// SIMATIC S7-200 SMART project (STEP 7-Micro/WIN SMART), CPU ST60

SYMBOL_TABLE V区符号
参数传输成功           V0.0     // 接收工控机传来的数据传输成功信号
参数是否更新           V0.1
挡板自动控制完成标志       V0.2
挡板电机开关           V0.3
挡板手动向内           V0.4
挡板手动向外           V0.5
置工件就绪            V1000.0
下料电机开关           V0.7
下料前进点动           V1.0
下料后退点动           V1.1
冷却电机开关           V1.2
冷却电机点动向内         V1.3
冷却电机点动向外         V1.4
挡板电机手动运行         V10.0
冷却电机手动运行         V10.1
下料电机手动运行         V10.2
挡板手动一键调节         V10.3
挡板一键调节完成标志       V10.4
挡板点动向内           V10.5
挡板点动向外           V10.6
挡板电机查找原点按钮       V11.1
下料电机查找原点按钮       V11.2
冷却电机查找原点按钮       V11.3
挡板自动控制           V11.4
下料下移一个工位         V11.5
下料启动按钮           V11.6
下料手动完成标志         V11.7
回到底部             V12.0
冷却自动控制           V12.1
挡板电机查找原点         V12.2
下料电机查找原点         V12.3
冷却电机查找原点         V12.4
冷却点动向内           V12.5
冷却点动向外           V12.6
挡板电机函数完成标志位      V20.1
挡板电机当前运动方向       V20.2
挡板电机查找原点完成位      V20.3
挡板电机GOTO完成位      V20.4
挡板电机错误参数         VB21
挡板电机当前位置         VD24
挡板电机当前速度         VD28
挡板电机移动位置         VD44
挡板电机速度           VD48
挡板电机移动模式         VB41
挡板电机停止运动轴        V40.1
挡板电机运动方向         V40.2
冷却电机初始化完成位       V60.1
冷却电机当前运动方向       V60.2
冷却电机查找原点完成位      V60.3
冷却电机GOTO完成位      V60.4
冷却电机错误参数         VB61
冷却电机当前位置         VD64
冷却电机当前速度         VD68
冷却电机移动位置         VD84
冷却电机速度           VD88
冷却电机移动模式         VB81
冷却电机停止运动轴        V80.1
冷却电机运动方向         V80.2
下料电机函数完成标志位      V100.1
下料电机当前运动方向       V100.2
下料电机查找原点完成位      V100.3
下料电机GOTO完成位      V100.4
下料电机错误参数         VB101
下料电机当前位置         VD104
下料电机当前速度         VD108
下料电机移动位置         VD124
下料电机速度           VD128
下料电机移动模式         VB121
下料电机停止运动轴        V120.1
下料电机运动方向         V120.2
下料电机运动到杆件放置      VD150
下料电机下移一个杆件位      VD154
下料电机一号杆件位置       VD158
下料电机二号杆件位置       VD162
下料电机三号杆件位置       VD166
下料电机四号杆件位置       VD170
下料电机五号杆件位置       VD174
下料电机运动到下料位置      VD178
上一杆件数据           VD140
当前杆件数据           VD144
轴0运动组态用          VB200    // VB200-VB292为轴0占用
轴1运动组态用          VB293    // VB293-VB385为轴1占用
轴2运动组态用          VB386    // VB386-VB478为轴2占用
链传动使能按钮          V400.0
链传动低速按钮          V400.1
链传动高速按钮          V400.2
链传动一个工位按钮        V400.3   // 链传动机构运动一个杆位按钮
链传动自动运行          V400.4
END_SYMBOL_TABLE

SYMBOL_TABLE 系统符号
Always_On        SM0.0    // 始终接通
First_Scan_On    SM0.1    // 仅在第一个扫描周期时接通
END_SYMBOL_TABLE

SYMBOL_TABLE M区符号
挡板超限报警           M0.0     // 挡板的位置超过左右极限传感器的位置
更新配对表            M0.1
电机是否就绪状态位        M0.3
上料步进到位状态位        M0.4
上料工件有无状态位        M0.5
下料步进到位状态位        M0.6
下料小车到位状态位        M0.7
步进报警信息           M1.0
上料传动故障报警         M1.1
两次杆件之差           MD12
END_SYMBOL_TABLE

SYMBOL_TABLE 定时器符号
顺序控制延时1          T33      // 短延时，保证正确读取到判断工件有无传感器的状态
顺序控制延时2          T34      // 短延时，保证正确读取到判断工件是否到位传感器的状态
顺序控制延时3          T35      // 短延时，保证正确读取到判断工件有无传感器的状态
上料故障报警定时         T37      // 设置定时，超时则报警
链传动控制定时器         T97
挡板运动脉冲1          T101     // 给一个运动脉冲信号，挡板移动到杆件长度处
下料运动脉冲1          T102     // 给一个运动脉冲信号，小车移动到机器人放料处
END_SYMBOL_TABLE

ORGANIZATION_BLOCK 主程序:OB1
TITLE=
BEGIN
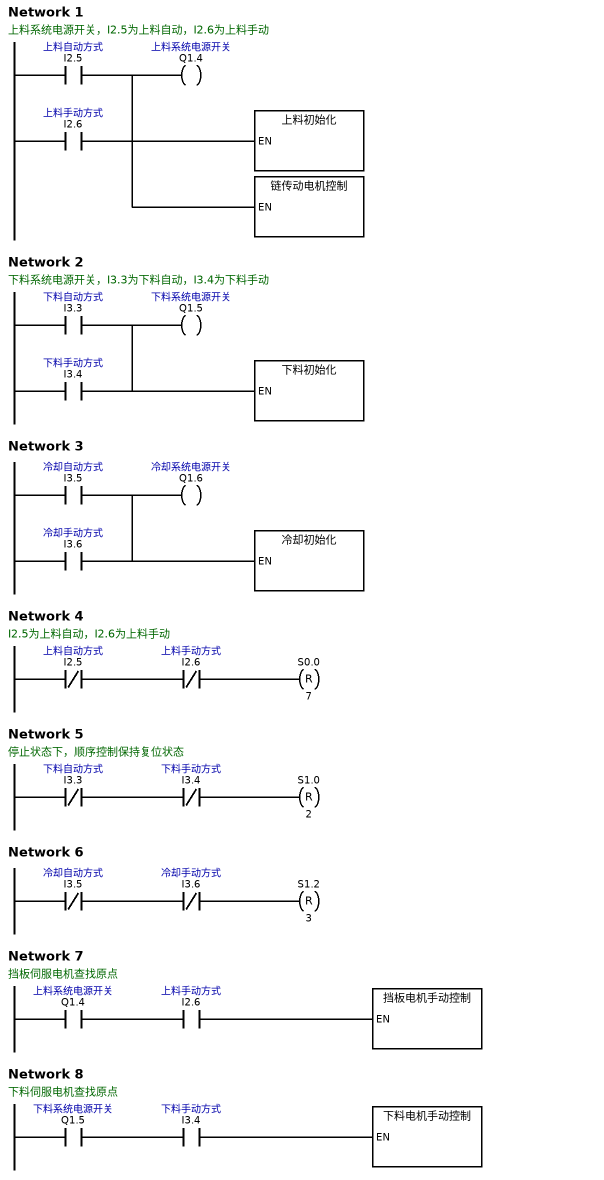
Network 1
// 上料系统电源开关，I2.5为上料自动，I2.6为上料手动
LD     上料自动方式:I2.5
O      上料手动方式:I2.6
=      上料系统电源开关:Q1.4
CALL   上料初始化:SBR14
CALL   链传动电机控制:SBR19
Network 2
// 下料系统电源开关，I3.3为下料自动，I3.4为下料手动
LD     下料自动方式:I3.3
O      下料手动方式:I3.4
=      下料系统电源开关:Q1.5
CALL   下料初始化:SBR15
Network 3
LD     冷却自动方式:I3.5
O      冷却手动方式:I3.6
=      冷却系统电源开关:Q1.6
CALL   冷却初始化:SBR16
Network 4
// I2.5为上料自动，I2.6为上料手动
LDN    上料自动方式:I2.5
AN     上料手动方式:I2.6
R      S0.0, 7
Network 5
// 停止状态下，顺序控制保持复位状态
LDN    下料自动方式:I3.3
AN     下料手动方式:I3.4
R      S1.0, 2
Network 6
LDN    冷却自动方式:I3.5
AN     冷却手动方式:I3.6
R      S1.2, 3
Network 7
// 挡板伺服电机查找原点
LD     上料系统电源开关:Q1.4
A      上料手动方式:I2.6
CALL   挡板电机手动控制:SBR7
Network 8
// 下料伺服电机查找原点
LD     下料系统电源开关:Q1.5
A      下料手动方式:I3.4
CALL   下料电机手动控制:SBR9
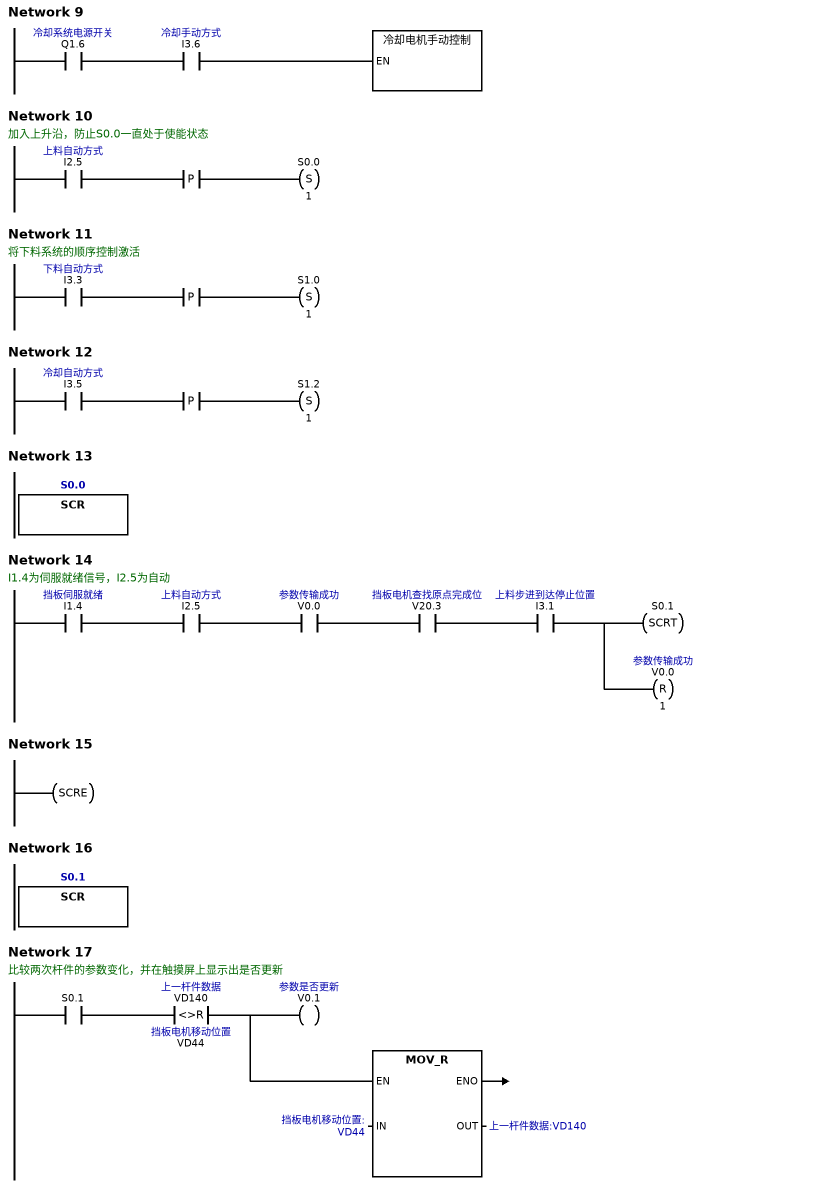
Network 9
LD     冷却系统电源开关:Q1.6
A      冷却手动方式:I3.6
CALL   冷却电机手动控制:SBR18
Network 10
// 加入上升沿，防止S0.0一直处于使能状态
LD     上料自动方式:I2.5
EU
S      S0.0, 1
Network 11
// 将下料系统的顺序控制激活
LD     下料自动方式:I3.3
EU
S      S1.0, 1
Network 12
LD     冷却自动方式:I3.5
EU
S      S1.2, 1
Network 13
LSCR   S0.0
Network 14
// I1.4为伺服就绪信号，I2.5为自动
LD     挡板伺服就绪:I1.4
A      上料自动方式:I2.5
A      参数传输成功:V0.0
A      挡板电机查找原点完成位:V20.3
A      上料步进到达停止位置:I3.1
SCRT   S0.1
R      参数传输成功:V0.0, 1
Network 15
SCRE
Network 16
LSCR   S0.1
Network 17
// 比较两次杆件的参数变化，并在触摸屏上显示出是否更新
LD     S0.1
AR<>   上一杆件数据:VD140, 挡板电机移动位置:VD44
=      参数是否更新:V0.1
MOVR   挡板电机移动位置:VD44, 上一杆件数据:VD140
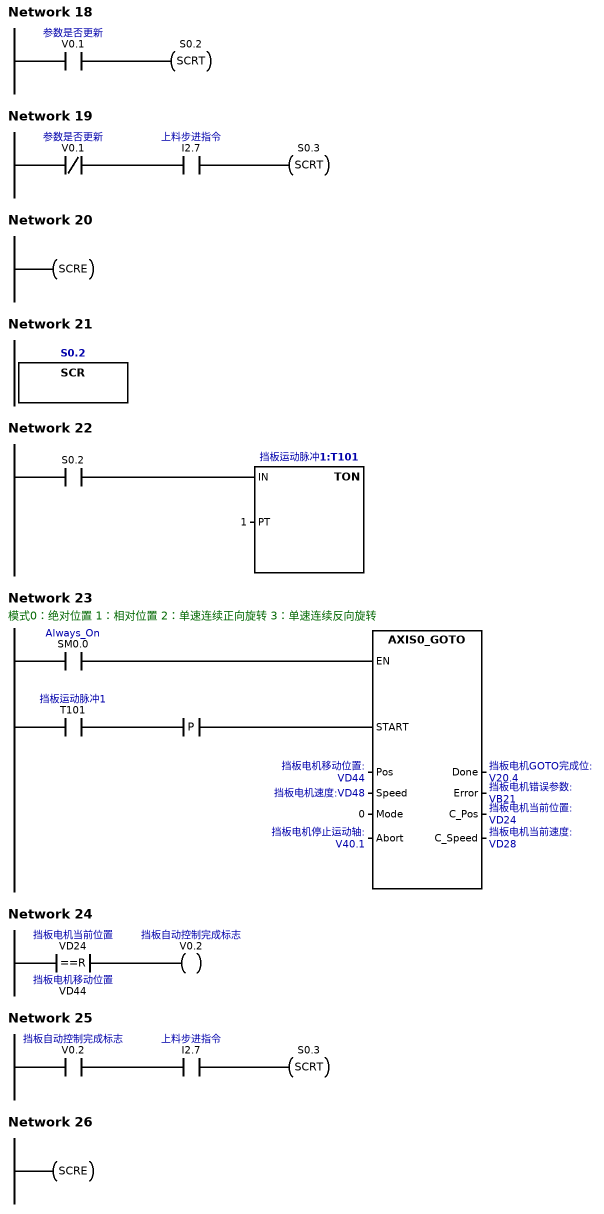
Network 18
LD     参数是否更新:V0.1
SCRT   S0.2
Network 19
LDN    参数是否更新:V0.1
A      上料步进指令:I2.7
SCRT   S0.3
Network 20
SCRE
Network 21
LSCR   S0.2
Network 22
LD     S0.2
TON    挡板运动脉冲1:T101, 1
Network 23
// 模式0：绝对位置 1：相对位置 2：单速连续正向旋转 3：单速连续反向旋转
LD     Always_On:SM0.0
=      L60.0
LD     挡板运动脉冲1:T101
EU
=      L63.7
LD     L60.0
CALL   AXIS0_GOTO:SBR2, L63.7, 挡板电机移动位置:VD44, 挡板电机速度:VD48, 0, 挡板电机停止运动轴:V40.1, 挡板电机GOTO完成位:V20.4, 挡板电机错误参数:VB21, 挡板电机当前位置:VD24, 挡板电机当前速度:VD28
Network 24
LDR=   挡板电机当前位置:VD24, 挡板电机移动位置:VD44
=      挡板自动控制完成标志:V0.2
Network 25
LD     挡板自动控制完成标志:V0.2
A      上料步进指令:I2.7
SCRT   S0.3
Network 26
SCRE
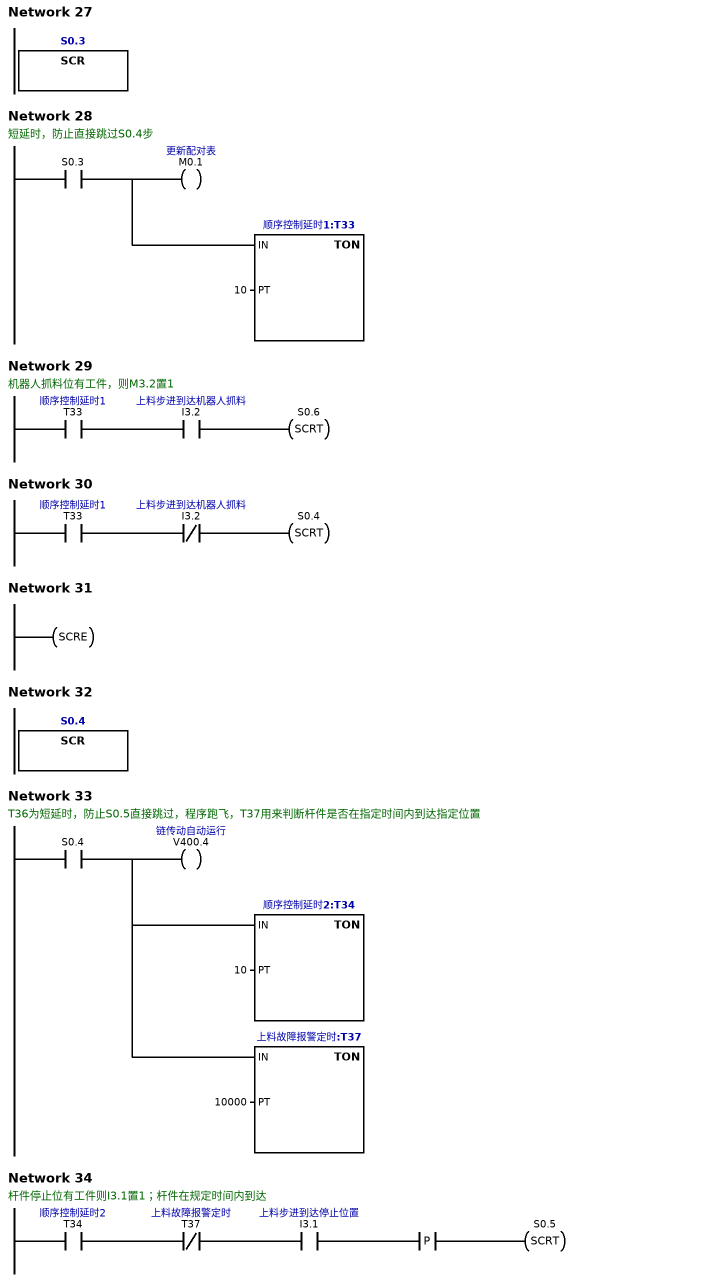
Network 27
LSCR   S0.3
Network 28
// 短延时，防止直接跳过S0.4步
LD     S0.3
=      更新配对表:M0.1
TON    顺序控制延时1:T33, 10
Network 29
// 机器人抓料位有工件，则M3.2置1
LD     顺序控制延时1:T33
A      上料步进到达机器人抓料:I3.2
SCRT   S0.6
Network 30
LD     顺序控制延时1:T33
AN     上料步进到达机器人抓料:I3.2
SCRT   S0.4
Network 31
SCRE
Network 32
LSCR   S0.4
Network 33
// T36为短延时，防止S0.5直接跳过，程序跑飞，T37用来判断杆件是否在指定时间内到达指定位置
LD     S0.4
=      链传动自动运行:V400.4
TON    顺序控制延时2:T34, 10
TON    上料故障报警定时:T37, 10000
Network 34
// 杆件停止位有工件则I3.1置1；杆件在规定时间内到达
LD     顺序控制延时2:T34
AN     上料故障报警定时:T37
A      上料步进到达停止位置:I3.1
EU
SCRT   S0.5
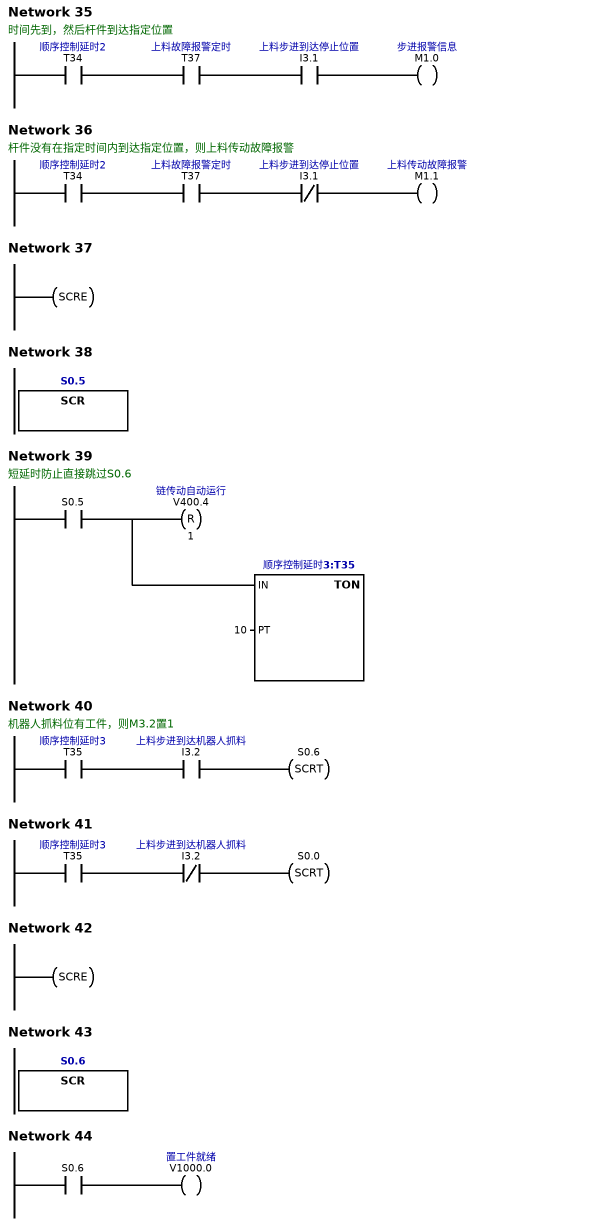
Network 35
// 时间先到，然后杆件到达指定位置
LD     顺序控制延时2:T34
A      上料故障报警定时:T37
A      上料步进到达停止位置:I3.1
=      步进报警信息:M1.0
Network 36
// 杆件没有在指定时间内到达指定位置，则上料传动故障报警
LD     顺序控制延时2:T34
A      上料故障报警定时:T37
AN     上料步进到达停止位置:I3.1
=      上料传动故障报警:M1.1
Network 37
SCRE
Network 38
LSCR   S0.5
Network 39
// 短延时防止直接跳过S0.6
LD     S0.5
R      链传动自动运行:V400.4, 1
TON    顺序控制延时3:T35, 10
Network 40
// 机器人抓料位有工件，则M3.2置1
LD     顺序控制延时3:T35
A      上料步进到达机器人抓料:I3.2
SCRT   S0.6
Network 41
LD     顺序控制延时3:T35
AN     上料步进到达机器人抓料:I3.2
SCRT   S0.0
Network 42
SCRE
Network 43
LSCR   S0.6
Network 44
LD     S0.6
=      置工件就绪:V1000.0
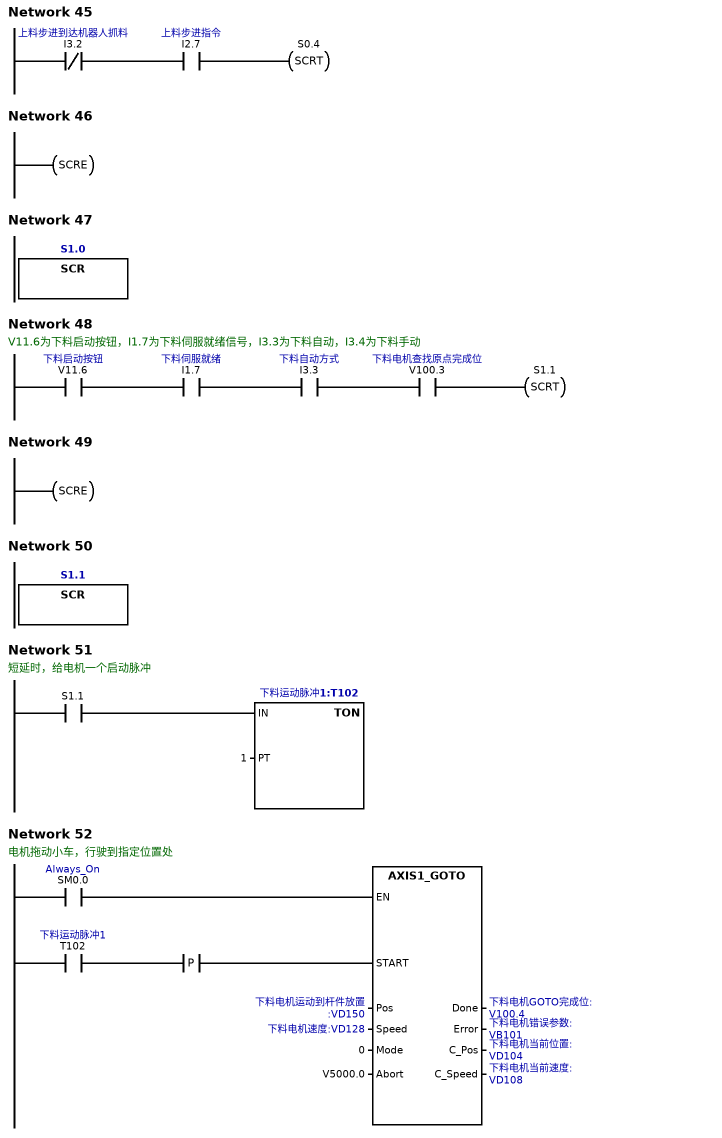
Network 45
LDN    上料步进到达机器人抓料:I3.2
A      上料步进指令:I2.7
SCRT   S0.4
Network 46
SCRE
Network 47
LSCR   S1.0
Network 48
// V11.6为下料启动按钮，I1.7为下料伺服就绪信号，I3.3为下料自动，I3.4为下料手动
LD     下料启动按钮:V11.6
A      下料伺服就绪:I1.7
A      下料自动方式:I3.3
A      下料电机查找原点完成位:V100.3
SCRT   S1.1
Network 49
SCRE
Network 50
LSCR   S1.1
Network 51
// 短延时，给电机一个启动脉冲
LD     S1.1
TON    下料运动脉冲1:T102, 1
Network 52
// 电机拖动小车，行驶到指定位置处
LD     Always_On:SM0.0
=      L60.0
LD     下料运动脉冲1:T102
EU
=      L63.7
LD     L60.0
CALL   AXIS1_GOTO:SBR6, L63.7, 下料电机运动到杆件放置:VD150, 下料电机速度:VD128, 0, V5000.0, 下料电机GOTO完成位:V100.4, 下料电机错误参数:VB101, 下料电机当前位置:VD104, 下料电机当前速度:VD108
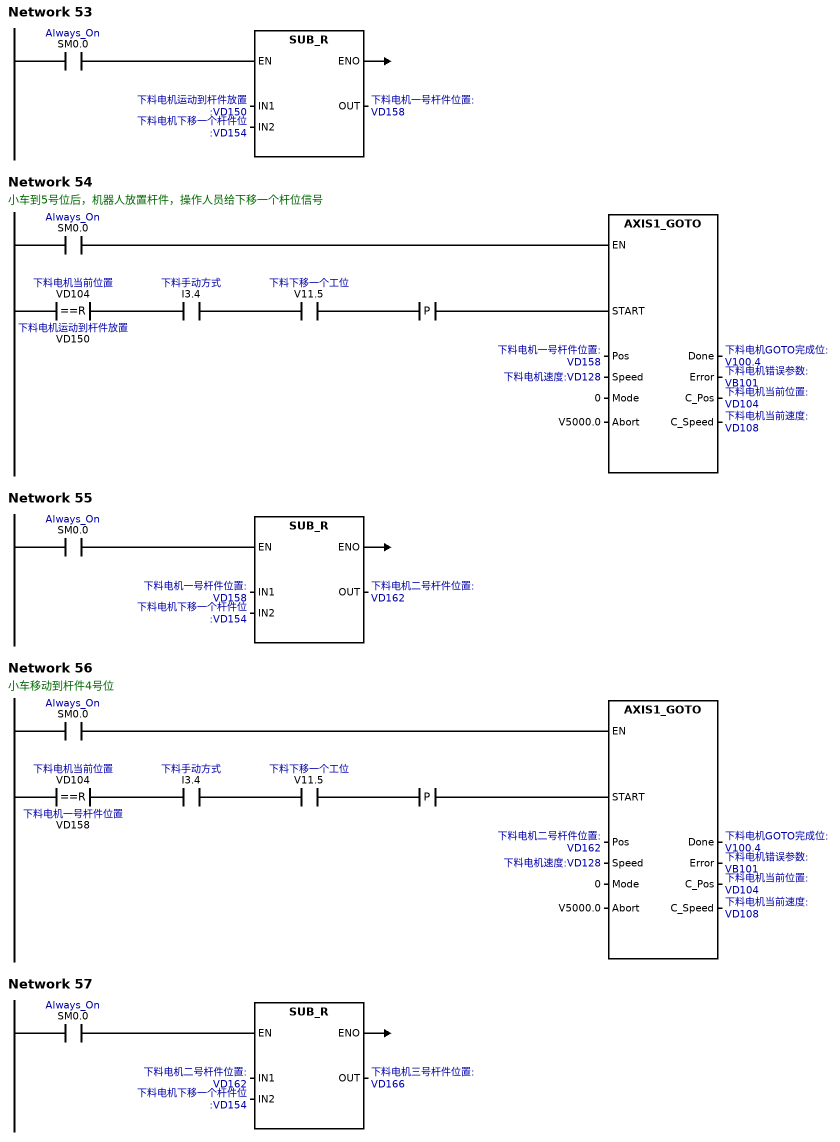
Network 53
LD     Always_On:SM0.0
MOVR   下料电机运动到杆件放置:VD150, 下料电机一号杆件位置:VD158
-R     下料电机下移一个杆件位:VD154, 下料电机一号杆件位置:VD158
Network 54
// 小车到5号位后，机器人放置杆件，操作人员给下移一个杆位信号
LD     Always_On:SM0.0
=      L60.0
LDR=   下料电机当前位置:VD104, 下料电机运动到杆件放置:VD150
A      下料手动方式:I3.4
A      下料下移一个工位:V11.5
EU
=      L63.7
LD     L60.0
CALL   AXIS1_GOTO:SBR6, L63.7, 下料电机一号杆件位置:VD158, 下料电机速度:VD128, 0, V5000.0, 下料电机GOTO完成位:V100.4, 下料电机错误参数:VB101, 下料电机当前位置:VD104, 下料电机当前速度:VD108
Network 55
LD     Always_On:SM0.0
MOVR   下料电机一号杆件位置:VD158, 下料电机二号杆件位置:VD162
-R     下料电机下移一个杆件位:VD154, 下料电机二号杆件位置:VD162
Network 56
// 小车移动到杆件4号位
LD     Always_On:SM0.0
=      L60.0
LDR=   下料电机当前位置:VD104, 下料电机一号杆件位置:VD158
A      下料手动方式:I3.4
A      下料下移一个工位:V11.5
EU
=      L63.7
LD     L60.0
CALL   AXIS1_GOTO:SBR6, L63.7, 下料电机二号杆件位置:VD162, 下料电机速度:VD128, 0, V5000.0, 下料电机GOTO完成位:V100.4, 下料电机错误参数:VB101, 下料电机当前位置:VD104, 下料电机当前速度:VD108
Network 57
LD     Always_On:SM0.0
MOVR   下料电机二号杆件位置:VD162, 下料电机三号杆件位置:VD166
-R     下料电机下移一个杆件位:VD154, 下料电机三号杆件位置:VD166
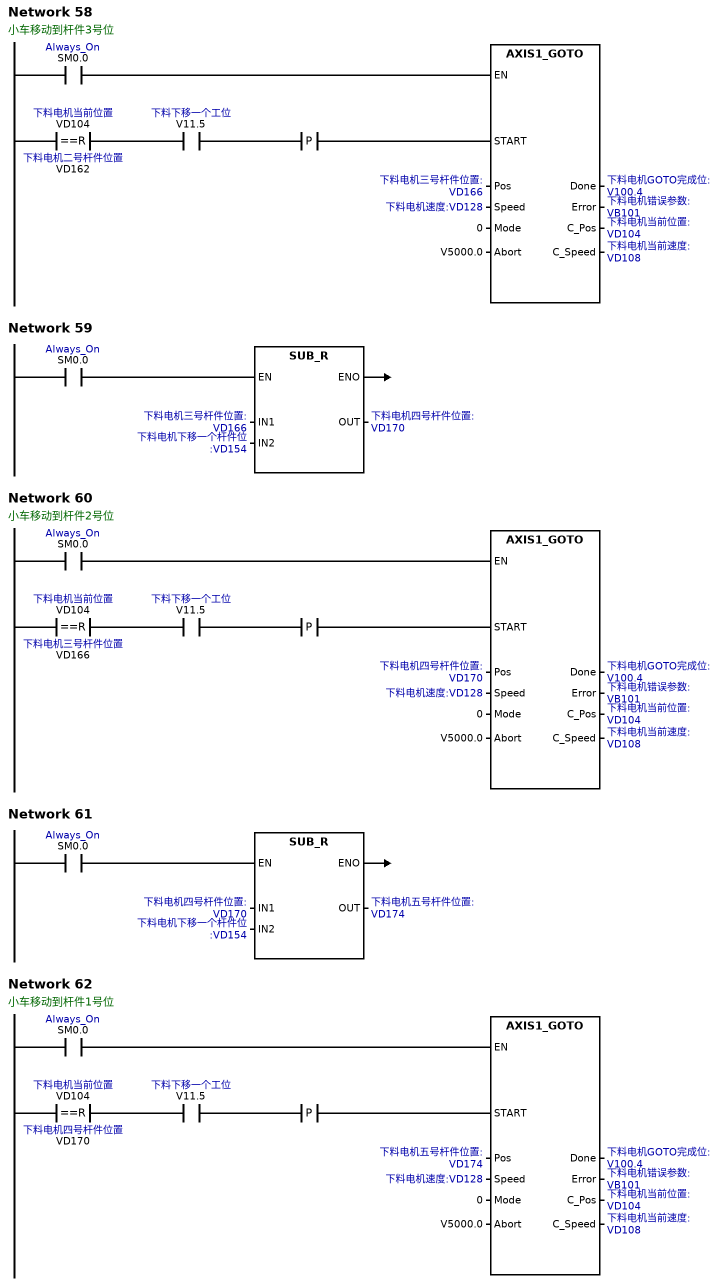
Network 58
// 小车移动到杆件3号位
LD     Always_On:SM0.0
=      L60.0
LDR=   下料电机当前位置:VD104, 下料电机二号杆件位置:VD162
A      下料下移一个工位:V11.5
EU
=      L63.7
LD     L60.0
CALL   AXIS1_GOTO:SBR6, L63.7, 下料电机三号杆件位置:VD166, 下料电机速度:VD128, 0, V5000.0, 下料电机GOTO完成位:V100.4, 下料电机错误参数:VB101, 下料电机当前位置:VD104, 下料电机当前速度:VD108
Network 59
LD     Always_On:SM0.0
MOVR   下料电机三号杆件位置:VD166, 下料电机四号杆件位置:VD170
-R     下料电机下移一个杆件位:VD154, 下料电机四号杆件位置:VD170
Network 60
// 小车移动到杆件2号位
LD     Always_On:SM0.0
=      L60.0
LDR=   下料电机当前位置:VD104, 下料电机三号杆件位置:VD166
A      下料下移一个工位:V11.5
EU
=      L63.7
LD     L60.0
CALL   AXIS1_GOTO:SBR6, L63.7, 下料电机四号杆件位置:VD170, 下料电机速度:VD128, 0, V5000.0, 下料电机GOTO完成位:V100.4, 下料电机错误参数:VB101, 下料电机当前位置:VD104, 下料电机当前速度:VD108
Network 61
LD     Always_On:SM0.0
MOVR   下料电机四号杆件位置:VD170, 下料电机五号杆件位置:VD174
-R     下料电机下移一个杆件位:VD154, 下料电机五号杆件位置:VD174
Network 62
// 小车移动到杆件1号位
LD     Always_On:SM0.0
=      L60.0
LDR=   下料电机当前位置:VD104, 下料电机四号杆件位置:VD170
A      下料下移一个工位:V11.5
EU
=      L63.7
LD     L60.0
CALL   AXIS1_GOTO:SBR6, L63.7, 下料电机五号杆件位置:VD174, 下料电机速度:VD128, 0, V5000.0, 下料电机GOTO完成位:V100.4, 下料电机错误参数:VB101, 下料电机当前位置:VD104, 下料电机当前速度:VD108
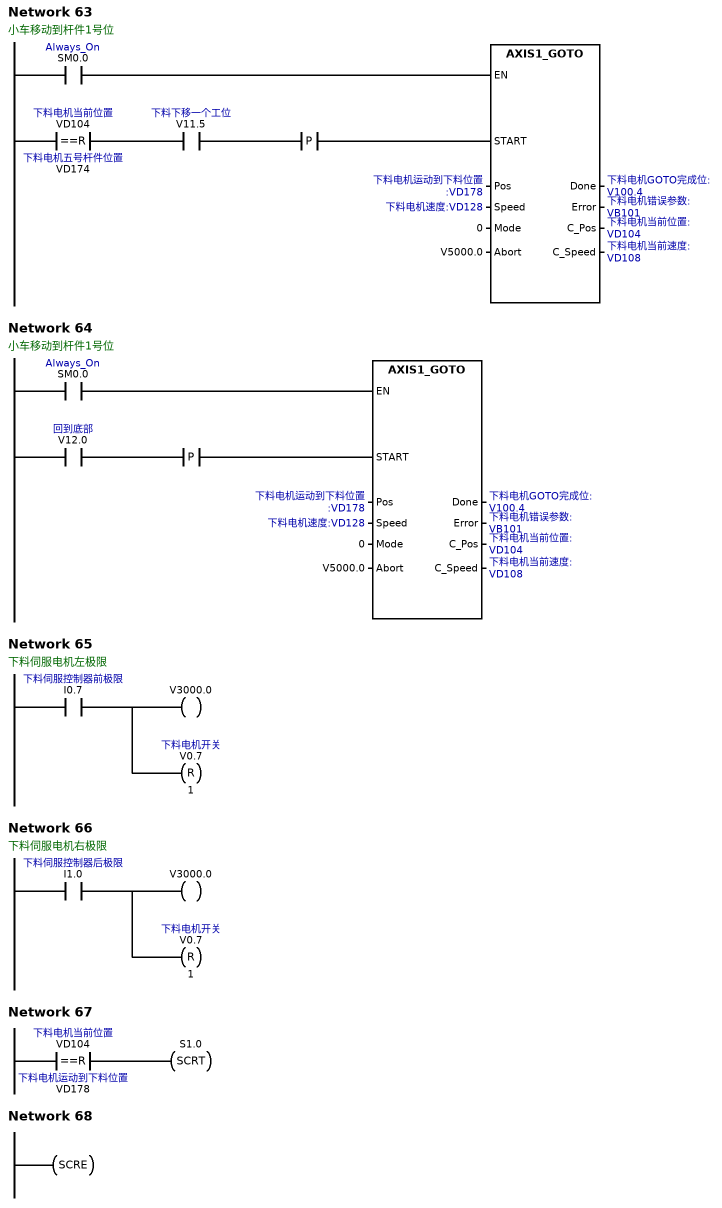
Network 63
// 小车移动到杆件1号位
LD     Always_On:SM0.0
=      L60.0
LDR=   下料电机当前位置:VD104, 下料电机五号杆件位置:VD174
A      下料下移一个工位:V11.5
EU
=      L63.7
LD     L60.0
CALL   AXIS1_GOTO:SBR6, L63.7, 下料电机运动到下料位置:VD178, 下料电机速度:VD128, 0, V5000.0, 下料电机GOTO完成位:V100.4, 下料电机错误参数:VB101, 下料电机当前位置:VD104, 下料电机当前速度:VD108
Network 64
// 小车移动到杆件1号位
LD     Always_On:SM0.0
=      L60.0
LD     回到底部:V12.0
EU
=      L63.7
LD     L60.0
CALL   AXIS1_GOTO:SBR6, L63.7, 下料电机运动到下料位置:VD178, 下料电机速度:VD128, 0, V5000.0, 下料电机GOTO完成位:V100.4, 下料电机错误参数:VB101, 下料电机当前位置:VD104, 下料电机当前速度:VD108
Network 65
// 下料伺服电机左极限
LD     下料伺服控制器前极限:I0.7
=      V3000.0
R      下料电机开关:V0.7, 1
Network 66
// 下料伺服电机右极限
LD     下料伺服控制器后极限:I1.0
=      V3000.0
R      下料电机开关:V0.7, 1
Network 67
LDR=   下料电机当前位置:VD104, 下料电机运动到下料位置:VD178
SCRT   S1.0
Network 68
SCRE
END_ORGANIZATION_BLOCK

// SBR0: protected block, not included

// SBR1: protected block, not included

// SBR2: protected block, not included

// SBR3: protected block, not included

// SBR4: protected block, not included

// SBR5: protected block, not included

// SBR6: protected block, not included

SUBROUTINE_BLOCK 挡板电机手动控制:SBR7
TITLE=子程序注释
BEGIN
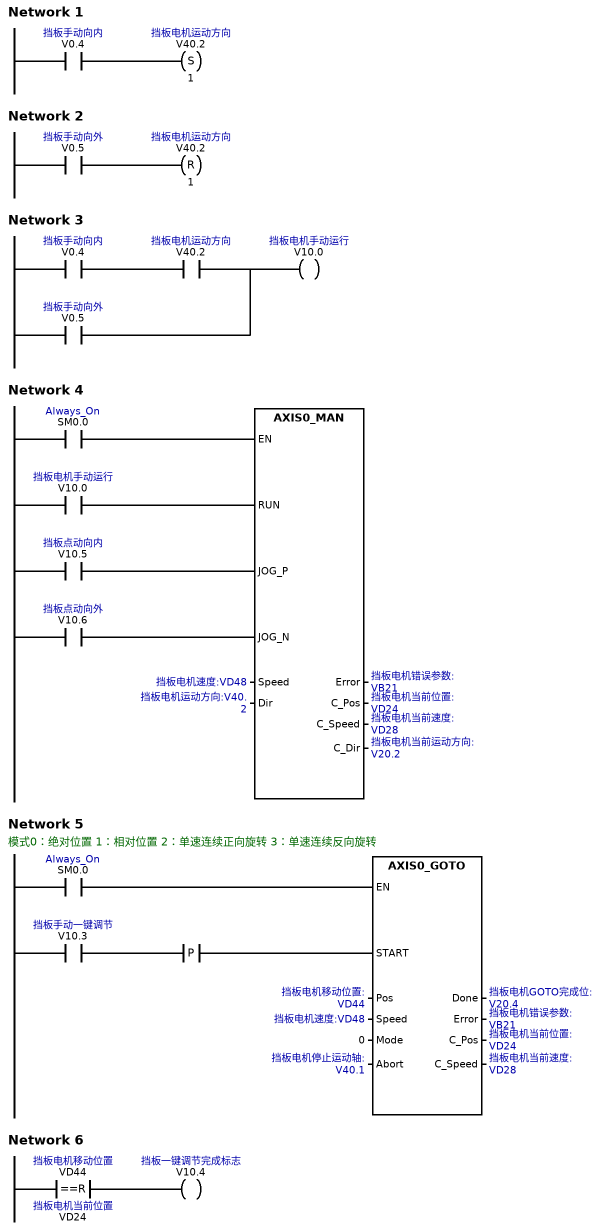
Network 1
LD     挡板手动向内:V0.4
S      挡板电机运动方向:V40.2, 1
Network 2
LD     挡板手动向外:V0.5
R      挡板电机运动方向:V40.2, 1
Network 3
LD     挡板手动向内:V0.4
A      挡板电机运动方向:V40.2
O      挡板手动向外:V0.5
=      挡板电机手动运行:V10.0
Network 4
LD     Always_On:SM0.0
=      L60.0
LD     挡板电机手动运行:V10.0
=      L63.7
LD     挡板点动向内:V10.5
=      L63.6
LD     挡板点动向外:V10.6
=      L63.5
LD     L60.0
CALL   AXIS0_MAN:SBR1, L63.7, L63.6, L63.5, 挡板电机速度:VD48, 挡板电机运动方向:V40.2, 挡板电机错误参数:VB21, 挡板电机当前位置:VD24, 挡板电机当前速度:VD28, 挡板电机当前运动方向:V20.2
Network 5
// 模式0：绝对位置 1：相对位置 2：单速连续正向旋转 3：单速连续反向旋转
LD     Always_On:SM0.0
=      L60.0
LD     挡板手动一键调节:V10.3
EU
=      L63.7
LD     L60.0
CALL   AXIS0_GOTO:SBR2, L63.7, 挡板电机移动位置:VD44, 挡板电机速度:VD48, 0, 挡板电机停止运动轴:V40.1, 挡板电机GOTO完成位:V20.4, 挡板电机错误参数:VB21, 挡板电机当前位置:VD24, 挡板电机当前速度:VD28
Network 6
LDR=   挡板电机移动位置:VD44, 挡板电机当前位置:VD24
=      挡板一键调节完成标志:V10.4
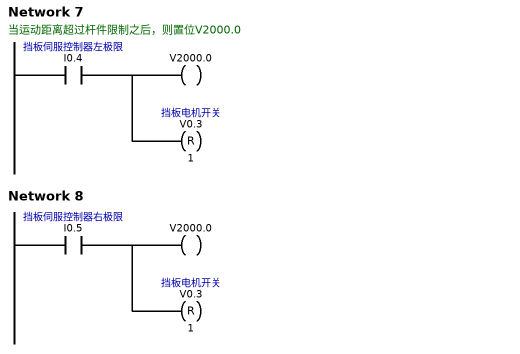
Network 7
// 当运动距离超过杆件限制之后，则置位V2000.0
LD     挡板伺服控制器左极限:I0.4
=      V2000.0
R      挡板电机开关:V0.3, 1
Network 8
LD     挡板伺服控制器右极限:I0.5
=      V2000.0
R      挡板电机开关:V0.3, 1
END_SUBROUTINE_BLOCK

// SBR8: protected block, not included

SUBROUTINE_BLOCK 下料电机手动控制:SBR9
TITLE=子程序注释
BEGIN
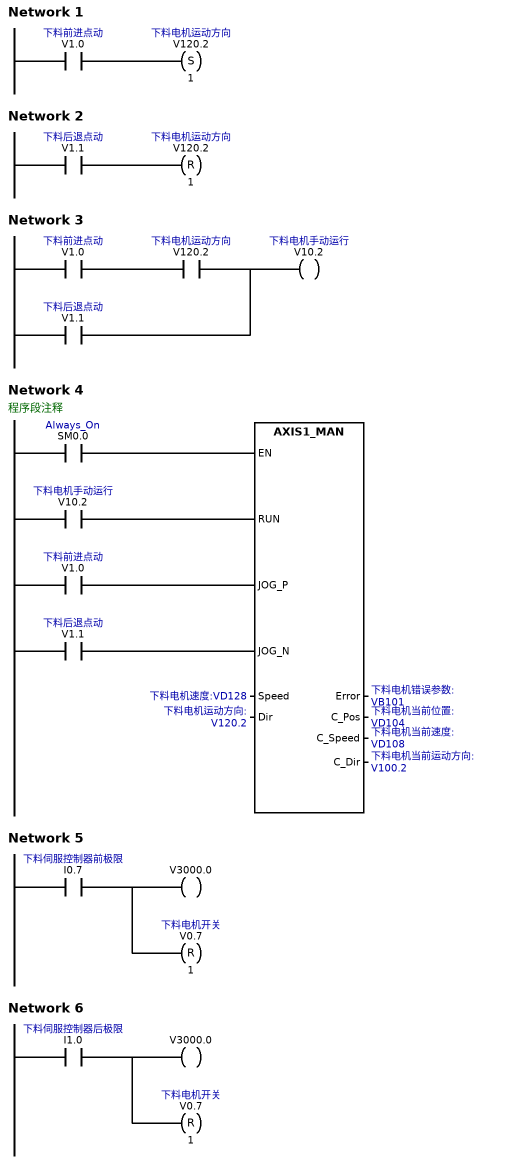
Network 1
LD     下料前进点动:V1.0
S      下料电机运动方向:V120.2, 1
Network 2
LD     下料后退点动:V1.1
R      下料电机运动方向:V120.2, 1
Network 3
LD     下料前进点动:V1.0
A      下料电机运动方向:V120.2
O      下料后退点动:V1.1
=      下料电机手动运行:V10.2
Network 4
// 程序段注释
LD     Always_On:SM0.0
=      L60.0
LD     下料电机手动运行:V10.2
=      L63.7
LD     下料前进点动:V1.0
=      L63.6
LD     下料后退点动:V1.1
=      L63.5
LD     L60.0
CALL   AXIS1_MAN:SBR5, L63.7, L63.6, L63.5, 下料电机速度:VD128, 下料电机运动方向:V120.2, 下料电机错误参数:VB101, 下料电机当前位置:VD104, 下料电机当前速度:VD108, 下料电机当前运动方向:V100.2
Network 5
LD     下料伺服控制器前极限:I0.7
=      V3000.0
R      下料电机开关:V0.7, 1
Network 6
LD     下料伺服控制器后极限:I1.0
=      V3000.0
R      下料电机开关:V0.7, 1
END_SUBROUTINE_BLOCK

// SBR10: protected block, not included

// SBR11: protected block, not included

// SBR12: protected block, not included

// SBR13: protected block, not included

SUBROUTINE_BLOCK 上料初始化:SBR14
TITLE=子程序注释
BEGIN
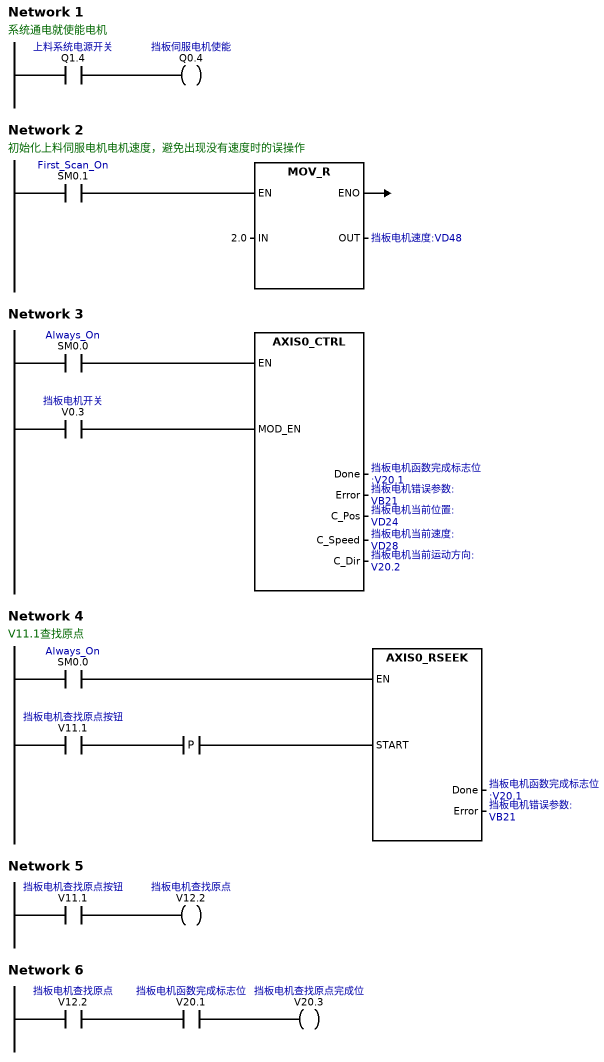
Network 1
// 系统通电就使能电机
LD     上料系统电源开关:Q1.4
=      挡板伺服电机使能:Q0.4
Network 2
// 初始化上料伺服电机电机速度，避免出现没有速度时的误操作
LD     First_Scan_On:SM0.1
MOVR   2.0, 挡板电机速度:VD48
Network 3
LD     Always_On:SM0.0
=      L60.0
LD     挡板电机开关:V0.3
=      L63.7
LD     L60.0
CALL   AXIS0_CTRL:SBR0, L63.7, 挡板电机函数完成标志位:V20.1, 挡板电机错误参数:VB21, 挡板电机当前位置:VD24, 挡板电机当前速度:VD28, 挡板电机当前运动方向:V20.2
Network 4
// V11.1查找原点
LD     Always_On:SM0.0
=      L60.0
LD     挡板电机查找原点按钮:V11.1
EU
=      L63.7
LD     L60.0
CALL   AXIS0_RSEEK:SBR3, L63.7, 挡板电机函数完成标志位:V20.1, 挡板电机错误参数:VB21
Network 5
LD     挡板电机查找原点按钮:V11.1
=      挡板电机查找原点:V12.2
Network 6
LD     挡板电机查找原点:V12.2
A      挡板电机函数完成标志位:V20.1
=      挡板电机查找原点完成位:V20.3
END_SUBROUTINE_BLOCK

SUBROUTINE_BLOCK 下料初始化:SBR15
TITLE=子程序注释
BEGIN
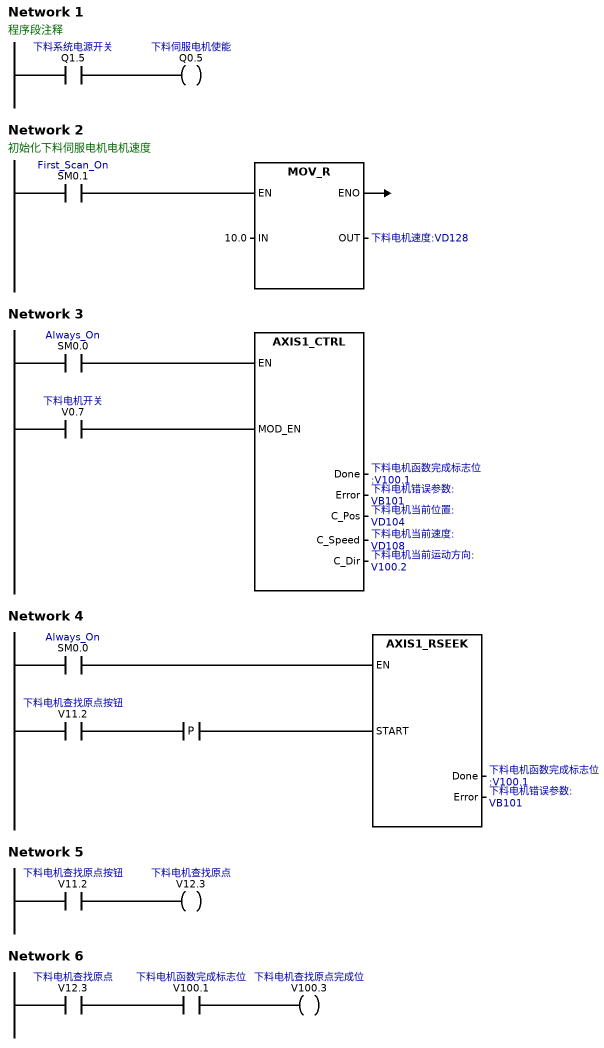
Network 1
// 程序段注释
LD     下料系统电源开关:Q1.5
=      下料伺服电机使能:Q0.5
Network 2
// 初始化下料伺服电机电机速度
LD     First_Scan_On:SM0.1
MOVR   10.0, 下料电机速度:VD128
Network 3
LD     Always_On:SM0.0
=      L60.0
LD     下料电机开关:V0.7
=      L63.7
LD     L60.0
CALL   AXIS1_CTRL:SBR4, L63.7, 下料电机函数完成标志位:V100.1, 下料电机错误参数:VB101, 下料电机当前位置:VD104, 下料电机当前速度:VD108, 下料电机当前运动方向:V100.2
Network 4
LD     Always_On:SM0.0
=      L60.0
LD     下料电机查找原点按钮:V11.2
EU
=      L63.7
LD     L60.0
CALL   AXIS1_RSEEK:SBR8, L63.7, 下料电机函数完成标志位:V100.1, 下料电机错误参数:VB101
Network 5
LD     下料电机查找原点按钮:V11.2
=      下料电机查找原点:V12.3
Network 6
LD     下料电机查找原点:V12.3
A      下料电机函数完成标志位:V100.1
=      下料电机查找原点完成位:V100.3
END_SUBROUTINE_BLOCK

SUBROUTINE_BLOCK 冷却初始化:SBR16
TITLE=子程序注释
BEGIN
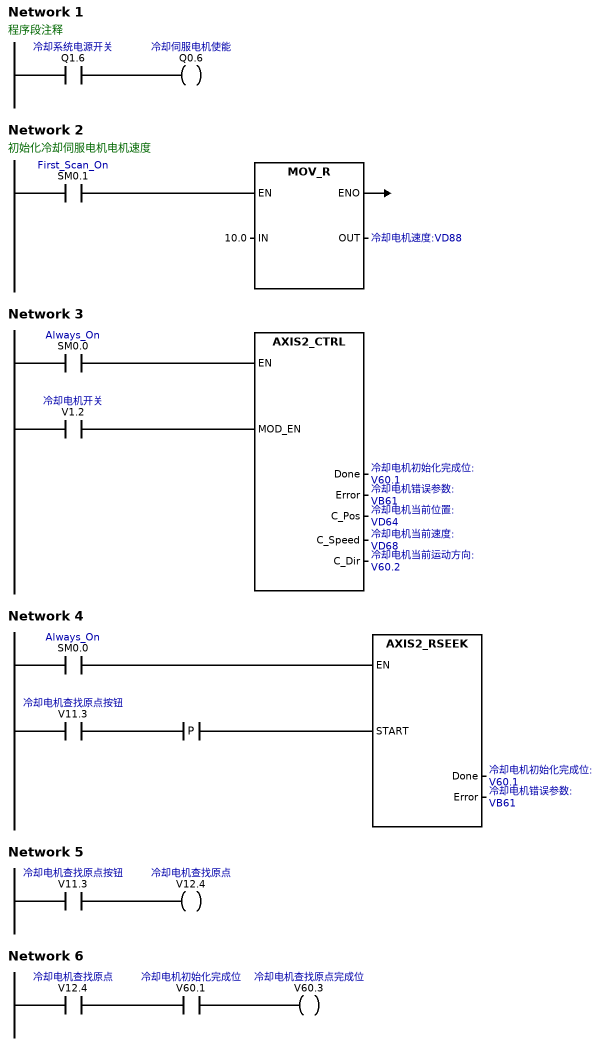
Network 1
// 程序段注释
LD     冷却系统电源开关:Q1.6
=      冷却伺服电机使能:Q0.6
Network 2
// 初始化冷却伺服电机电机速度
LD     First_Scan_On:SM0.1
MOVR   10.0, 冷却电机速度:VD88
Network 3
LD     Always_On:SM0.0
=      L60.0
LD     冷却电机开关:V1.2
=      L63.7
LD     L60.0
CALL   AXIS2_CTRL:SBR10, L63.7, 冷却电机初始化完成位:V60.1, 冷却电机错误参数:VB61, 冷却电机当前位置:VD64, 冷却电机当前速度:VD68, 冷却电机当前运动方向:V60.2
Network 4
LD     Always_On:SM0.0
=      L60.0
LD     冷却电机查找原点按钮:V11.3
EU
=      L63.7
LD     L60.0
CALL   AXIS2_RSEEK:SBR13, L63.7, 冷却电机初始化完成位:V60.1, 冷却电机错误参数:VB61
Network 5
LD     冷却电机查找原点按钮:V11.3
=      冷却电机查找原点:V12.4
Network 6
LD     冷却电机查找原点:V12.4
A      冷却电机初始化完成位:V60.1
=      冷却电机查找原点完成位:V60.3
END_SUBROUTINE_BLOCK

SUBROUTINE_BLOCK 冷却电机手动控制:SBR18
TITLE=子程序注释
BEGIN
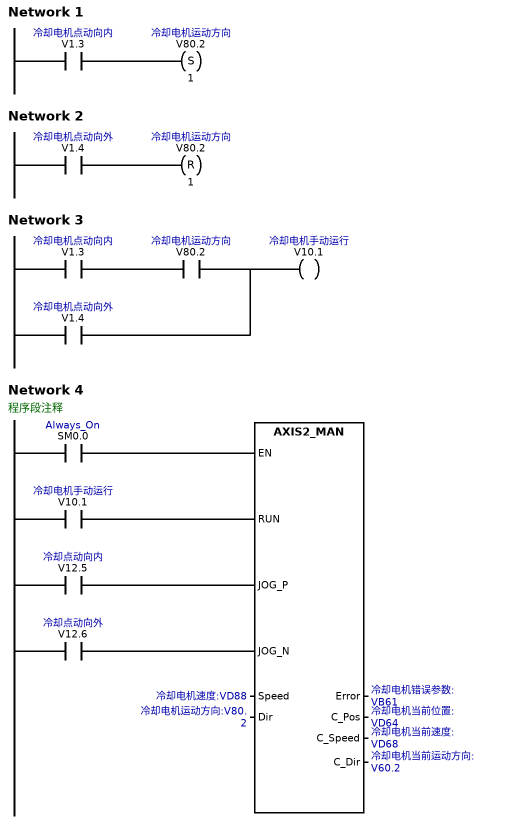
Network 1
LD     冷却电机点动向内:V1.3
S      冷却电机运动方向:V80.2, 1
Network 2
LD     冷却电机点动向外:V1.4
R      冷却电机运动方向:V80.2, 1
Network 3
LD     冷却电机点动向内:V1.3
A      冷却电机运动方向:V80.2
O      冷却电机点动向外:V1.4
=      冷却电机手动运行:V10.1
Network 4
// 程序段注释
LD     Always_On:SM0.0
=      L60.0
LD     冷却电机手动运行:V10.1
=      L63.7
LD     冷却点动向内:V12.5
=      L63.6
LD     冷却点动向外:V12.6
=      L63.5
LD     L60.0
CALL   AXIS2_MAN:SBR11, L63.7, L63.6, L63.5, 冷却电机速度:VD88, 冷却电机运动方向:V80.2, 冷却电机错误参数:VB61, 冷却电机当前位置:VD64, 冷却电机当前速度:VD68, 冷却电机当前运动方向:V60.2
END_SUBROUTINE_BLOCK

SUBROUTINE_BLOCK 链传动电机控制:SBR19
TITLE=子程序注释
BEGIN
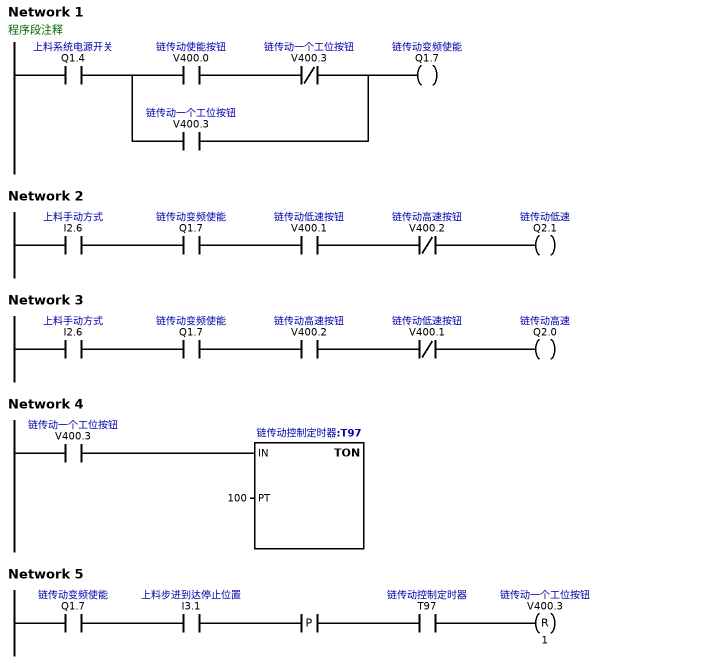
Network 1
// 程序段注释
LD     上料系统电源开关:Q1.4
LD     链传动使能按钮:V400.0
AN     链传动一个工位按钮:V400.3
O      链传动一个工位按钮:V400.3
ALD
=      链传动变频使能:Q1.7
Network 2
LD     上料手动方式:I2.6
A      链传动变频使能:Q1.7
A      链传动低速按钮:V400.1
AN     链传动高速按钮:V400.2
=      链传动低速:Q2.1
Network 3
LD     上料手动方式:I2.6
A      链传动变频使能:Q1.7
A      链传动高速按钮:V400.2
AN     链传动低速按钮:V400.1
=      链传动高速:Q2.0
Network 4
LD     链传动一个工位按钮:V400.3
TON    链传动控制定时器:T97, 100
Network 5
LD     链传动变频使能:Q1.7
A      上料步进到达停止位置:I3.1
EU
A      链传动控制定时器:T97
R      链传动一个工位按钮:V400.3, 1
END_SUBROUTINE_BLOCK
